Fanuc KAREL source: kt00983.KL

-- PROVISIONAL review KL for V770-1; original PC SHA256 11da83909a2230dcc4315e0d5bca70873cc57d8cc4d134eec3d9b3b17bf03ed2
-- Incomplete behavior may be omitted. Consult companion uncertainty JSON. Do not deploy.
PROGRAM KT00983
%NOLOCKGROUP
VAR
  R1 : REAL
  R2 : REAL
-- UNRESOLVED_DECL CFG type=00001c
-- UNRESOLVED_DECL OUT type=000102
BEGIN
  -- UNRESOLVED_PC offsets 5-16; opcodes 2E,23
  -- UNRESOLVED_PC offsets 21-32; opcodes 2E,23
  -- UNRESOLVED_PC offsets 37-48; opcodes 2E,23
  -- UNRESOLVED_PC offsets 53-64; opcodes 2E,23
  -- UNRESOLVED_PC offsets 69-79; opcodes 9D,22,A5
  -- UNRESOLVED_PC offsets 84-141; opcodes 27,22,22,22,22,22,22,22,76,7E,4A
  -- UNRESOLVED_PC offsets 146-150; opcodes 7F
END KT00983
